FUNCTION_BLOCK LE_BOOL (* IEC 61131-3,Table 28#8 *)
  (* Standard: 61131-3 *)
  (* Version 0.0, 2004-12-15, JHC, Rockwell Automation, Converted from SRC format. *)
  (* Compiler header: package fb.rt.plc.comp; *)
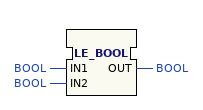
  VAR_INPUT
    IN1 : BOOL;
    IN2 : BOOL;
  END_VAR
  VAR_OUTPUT
    OUT : BOOL;
  END_VAR
END_FUNCTION_BLOCK
